(* PLC project cmd_motor_2d2s, Dassault Systèmes ControlBuild 2024x *)
(* stored: creationDateTime 2023-10-03T11:13:35-01:00 *)

FUNCTION_BLOCK actuator
  VAR_INPUT
    autoMode : BOOL := false;
    manualMode : BOOL := false;
  END_VAR
  VAR_INPUT
    autoFwdCmd : BOOL := false;
    autoBwdCmd : BOOL := false;
    autoHSCmd : BOOL := false;
    autoLSCmd : BOOL := false;
  END_VAR
  VAR_INPUT
    forwardPB : BOOL := false;
    backwardPB : BOOL := false;
    highSpeedPB : BOOL := false;
    lowSpeedPB : BOOL := false;
    stopPB : BOOL := false;
  END_VAR
  VAR_INPUT
    generalFault : BOOL := false;
  END_VAR
  VAR_OUTPUT
    forwardCmd : BOOL := false;
    backwardCmd : BOOL := false;
    highSpeedCmd : BOOL := false;
    lowSpeedCmd : BOOL := false;
  END_VAR

(* LD diagram, written out as Structured Text *)
1:
forwardCmd := (autoMode AND autoFwdCmd OR manualMode AND (forwardCmd OR forwardPB AND NOT backwardPB) AND NOT stopPB AND NOT backwardCmd) AND NOT generalFault;
2:
backwardCmd := (autoMode AND autoBwdCmd OR manualMode AND (backwardCmd OR backwardPB AND NOT forwardPB) AND NOT stopPB AND NOT forwardCmd) AND NOT generalFault;
3:
highSpeedCmd := (autoMode AND autoHSCmd OR manualMode AND (highSpeedPB OR highSpeedCmd) AND NOT lowSpeedPB) AND NOT generalFault;
lowSpeedCmd := (autoMode AND autoLSCmd OR manualMode AND (lowSpeedPB OR lowSpeedCmd) AND NOT highSpeedPB) AND NOT generalFault;
END_FUNCTION_BLOCK

FUNCTION_BLOCK faults
  VAR_INPUT
    forwardCmd : BOOL := false;
    backwardCmd : BOOL := false;
    highSpeedCmd : BOOL := false;
    lowSpeedCmd : BOOL := false;
  END_VAR
  VAR_INPUT
    thermalFB : BOOL := false;
    forwardFB : BOOL := false;
    backwardFB : BOOL := false;
    highSpeedFB : BOOL := false;
    lowSpeedFB : BOOL := false;
  END_VAR
  VAR_INPUT
    acknowledgePB : BOOL := false;
  END_VAR
  VAR_OUTPUT
    generalFault : BOOL := false;
  END_VAR
  VAR
    thermalFault : BOOL := false;
    forwardFBFault : BOOL := false;
    backwardFBFault : BOOL := false;
  END_VAR

(* LD diagram, written out as Structured Text *)
1:
IF acknowledgePB THEN thermalFault := FALSE; END_IF;
IF acknowledgePB THEN forwardFBFault := FALSE; END_IF;
IF acknowledgePB THEN backwardFBFault := FALSE; END_IF;
IF acknowledgePB THEN generalFault := FALSE; END_IF;
2:
IF TON_FW.Q0 AND (NOT forwardFB OR highSpeedCmd AND NOT highSpeedFB OR lowSpeedCmd AND NOT lowSpeedFB) THEN forwardFBFault := TRUE; END_IF;
IF TON_BW.Q0 AND (NOT backwardFB OR lowSpeedCmd AND NOT lowSpeedFB OR highSpeedCmd AND NOT highSpeedFB) THEN backwardFBFault := TRUE; END_IF;
3:
IF NOT thermalFB THEN thermalFault := TRUE; END_IF;
4:
IF thermalFault OR forwardFBFault OR backwardFBFault THEN generalFault := TRUE; END_IF;
TON_FW(IN := (highSpeedCmd OR lowSpeedCmd) AND forwardCmd, PT := T#0h0m2s0ms);
TON_BW(IN := (lowSpeedCmd OR highSpeedCmd) AND backwardCmd, PT := T#0h0m2s0ms);
END_FUNCTION_BLOCK

(* Command of a motor with two directions and two speeds and with fault detection *)
PROGRAM cmd_equipment_library.cmd_motor_2d2s
  VAR_INPUT
    autoMode : BOOL := false;
    manualMode : BOOL := false;
  END_VAR
  VAR_INPUT
    autoFwdCmd : BOOL := false;
    autoBwdCmd : BOOL := false;
    autoHSCmd : BOOL := false;
    autoLSCmd : BOOL := false;
  END_VAR
  VAR_INPUT
    forwardPB : BOOL := false;
    backwardPB : BOOL := false;
    highSpeedPB : BOOL := false;
    lowSpeedPB : BOOL := false;
    stopPB : BOOL := false;
  END_VAR
  VAR_INPUT
    forwardFB : BOOL := false;
    backwardFB : BOOL := false;
    highSpeedFB : BOOL := false;
    lowSpeedFB : BOOL := false;
    thermalFB : BOOL := false;
  END_VAR
  VAR_INPUT
    acknowledgePB : BOOL := false;
  END_VAR
  VAR_OUTPUT
    forwardCmd : BOOL := false;
    backwardCmd : BOOL := false;
    highSpeedCmd : BOOL := false;
    lowSpeedCmd : BOOL := false;
  END_VAR
  VAR_OUTPUT
    generalFault : BOOL := false;
  END_VAR

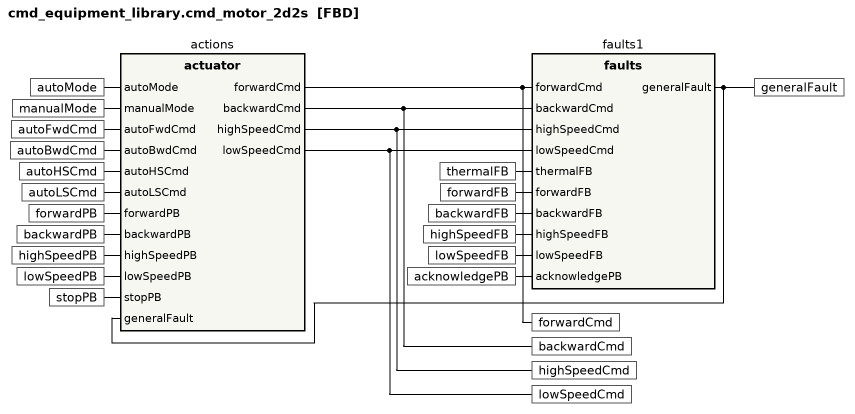
(* FBD diagram, written out as Structured Text *)
faults1(forwardCmd := actions.forwardCmd, backwardCmd := actions.backwardCmd, highSpeedCmd := actions.highSpeedCmd, lowSpeedCmd := actions.lowSpeedCmd, thermalFB := thermalFB, forwardFB := forwardFB, backwardFB := backwardFB, highSpeedFB := highSpeedFB, lowSpeedFB := lowSpeedFB, acknowledgePB := acknowledgePB);
actions(autoMode := autoMode, manualMode := manualMode, autoFwdCmd := autoFwdCmd, autoBwdCmd := autoBwdCmd, autoHSCmd := autoHSCmd, autoLSCmd := autoLSCmd, forwardPB := forwardPB, backwardPB := backwardPB, highSpeedPB := highSpeedPB, lowSpeedPB := lowSpeedPB, stopPB := stopPB, generalFault := faults1.generalFault);
forwardCmd := actions.forwardCmd;
backwardCmd := actions.backwardCmd;
highSpeedCmd := actions.highSpeedCmd;
lowSpeedCmd := actions.lowSpeedCmd;
generalFault := faults1.generalFault;
END_PROGRAM
